PROGRAM MAIN
VAR
	fbSequence : ControlFBD_Sequence;
	fbBlink    : BLINK;
	
	mxAutoRunOk: BOOL;
	mxAutoModeReady: BOOL;
	ixSliderAout: BOOL;
	ixDrillDown: BOOL;
	ixDrillUp: BOOL;
	ixSliderBout: BOOL;
	ixSliderBin: BOOL;
	
	mxAutoAout       : BOOL;
    mxAutoDrillDown: BOOL;
    mxAutoDrillUp    : BOOL;
    mxAutoBout       : BOOL;
    mxAutoBin        : BOOL;
    mxAutoAin        : BOOL;
	
END_VAR

ControlFBD();
(* Auto sequence engine *)
fbSequence(
   mxAutoRunOk     := ControlFBD.mxAutoRunOk,
    mxAutoModeReady := ControlFBD.mxAutoModeReady,
    ixSliderAout    := ControlFBD.ixSliderAout,
    ixDrillDown     := ControlFBD.ixDrillDown,
    ixDrillUp       := ControlFBD.ixDrillUp,
	ixSliderAin    := ControlFBD.ixSliderAin,
    ixSliderBout    := ControlFBD.ixSliderBout,
    ixSliderBin     := ControlFBD.ixSliderBin
);

ControlFBD.mxAutoAout := fbSequence.mxAutoAOut;
ControlFBD.mxAutoAin := fbSequence.mxAutoAIn;
ControlFBD.mxAutoBout := fbSequence.mxAutoBout;
ControlFBD.mxAutoBin := fbSequence.mxAutoBin;
ControlFBD.mxAutoDrillOut := fbSequence.mxAutoDrillDown;
ControlFBD.mxAutoDrillUp := fbSequence.mxAutoDrillUp;

fbBlink(
    OnTime := T#0.5S,
    OffTime := T#1S
);

END_PROGRAM

(* stored: Version 1.1.0.1
   POU MAIN: Id {54befd21-3517-4010-bc97-4f29dd46757e}, SpecialFunc None *)
